# EPICS autosave request: LabJackApp/Db/LabJackWaveformDig_settings.req
$(P)WaveDigNumPoints
$(P)WaveDigFirstChan
$(P)WaveDigNumChans
$(P)WaveDigDwell
$(P)WaveDigExtTrigger
$(P)WaveDigExtClock
$(P)WaveDigAutoRestart
$(P)WaveDigSettlingTime
$(P)WaveDigResolution
$(P)WaveDigReadWF.SCAN
